// TwinCAT 3 PLC project Untitled1
// ProgramVersion: 3.1.4020.10
// libraries:
//   Tc2_Standard, * (Beckhoff Automation GmbH)
//   Tc2_System, * (Beckhoff Automation GmbH)
//   Tc3_Module, * (Beckhoff Automation GmbH)
//   VisuDialogs, * (System)
// project tree:
//   / GlobalTextList.TcGTLO (not stored), PlcTask.TcTTO (not stored), Visualization Manager.TcVMO (not stored)
//   POUs/ FB_PIZZA_OVEN.TcPOU (not stored), FB_SIMPLE.TcPOU, MAIN.TcPOU (not stored)
//   VISUs/ Visualization_1.TcVIS (not stored)

// ---- POUs/FB_SIMPLE.TcPOU
FUNCTION_BLOCK FB_SIMPLE
VAR_INPUT
	bPizzaDone : BOOL;
END_VAR
VAR_OUTPUT
	bLightOn : BOOL;
END_VAR
VAR
END_VAR

IF bPizzaDone THEN
	bLightOn := TRUE;
ELSE
	bLightOn := FALSE;
END_IF

END_FUNCTION_BLOCK
